(* PLC project Untitled1, Beckhoff Automation GmbH TwinCAT PLC Control 3.5.10.30 *)
(* stored: creationDateTime 2020-09-30T13:14:05.8851775, modificationDateTime 2020-09-30T13:14:05.8881769 *)

TYPE enum_E :
(
	elit_gopickup,
	elit_init0,
	elit_init1,
	elit_init2,
	elit_init3,
	elit_init4,
	elit_init5,
	elit_init6,
	elit_init7,
	elit_init8,
	elit_init9,
	elit_init_error,
	elit_init_ok,
	elit_init_sensor_check,
	elit_initialized,
	elit_running,
	elit_starting,
	elit_wait_init,
	elit_wait_start
);
END_TYPE

TYPE STATE :
STRUCT
	curTime: LREAL;
	dvar_M_example_controller_a_x2distributing AT %Q*: BOOL;
	dvar_M_example_controller_a_zdown AT %Q*: BOOL;
	dvar_M_example_controller_count AT %Q*: DINT;
	dvar_M_example_controller AT %Q*: enum_E;
	dvar_M_HardwareMap_out_a_Dstartled AT %Q*: BOOL;
	dvar_M_HardwareMap_out_a_Dresetled AT %Q*: BOOL;
	dvar_M_HardwareMap_out_a_DledQ1 AT %Q*: BOOL;
	dvar_M_HardwareMap_out_a_DledQ2 AT %Q*: BOOL;
	dvar_M_HardwareMap_out_a_Dout4 AT %Q*: BOOL;
	dvar_M_HardwareMap_out_a_Dout5 AT %Q*: BOOL;
	dvar_M_HardwareMap_out_a_Dout6 AT %Q*: BOOL;
	dvar_M_HardwareMap_out_a_Dout7 AT %Q*: BOOL;
	dvar_M_HardwareMap_out_a_pusher1 AT %Q*: BOOL;
	dvar_M_HardwareMap_out_a_pusher2 AT %Q*: BOOL;
	dvar_M_HardwareMap_out_a_pusher3 AT %Q*: BOOL;
	dvar_M_HardwareMap_out_a_Hstartled AT %Q*: BOOL;
	dvar_M_HardwareMap_out_a_Hresetled AT %Q*: BOOL;
	dvar_M_HardwareMap_out_a_HledQ1 AT %Q*: BOOL;
	dvar_M_HardwareMap_out_a_HledQ2 AT %Q*: BOOL;
	dvar_M_HardwareMap_out_a_Hout4 AT %Q*: BOOL;
	dvar_M_HardwareMap_out_a_Hout5 AT %Q*: BOOL;
	dvar_M_HardwareMap_out_a_Hout6 AT %Q*: BOOL;
	dvar_M_HardwareMap_out_a_Hout7 AT %Q*: BOOL;
	dvar_M_HardwareMap_out_a_x2distributing AT %Q*: BOOL;
	dvar_M_HardwareMap_out_a_x2testing AT %Q*: BOOL;
	dvar_M_HardwareMap_out_a_zdown AT %Q*: BOOL;
	dvar_M_HardwareMap_out_a_gripperclose AT %Q*: BOOL;
	dvar_M_HardwareMap_out_a_transfer2pickpos AT %Q*: BOOL;
	dvar_M_HardwareMap_out_a_transfer2droppos AT %Q*: BOOL;
	dvar_M_HardwareMap_out_a_vacuum AT %Q*: BOOL;
	dvar_M_HardwareMap_out_a_ejectpulse AT %Q*: BOOL;
	dvar_M_HardwareMap_out_a_handlingready AT %Q*: BOOL;
	dvar_M_HardwareMap_init_err_sen_idx AT %Q*: DINT;
	dvar_M_HardwareMap_init_err_led_idx AT %Q*: DINT;
	cvar_M_HardwareMap_t AT %Q*: LREAL;
	dvar_M_HardwareMap AT %Q*: enum_E;
END_STRUCT
END_TYPE

(* global variable list INPUTS *)
VAR_GLOBAL
	ivar_s_Dstartbutton AT %I*: BOOL;
	ivar_s_Dstopbutton AT %I*: BOOL;
	ivar_s_Dresetbutton AT %I*: BOOL;
	ivar_s_Dautoswitch AT %I*: BOOL;
	ivar_s_pusher1_in AT %I*: BOOL;
	ivar_s_pusher1_out AT %I*: BOOL;
	ivar_s_stack1filled AT %I*: BOOL;
	ivar_s_product1 AT %I*: BOOL;
	ivar_s_pusher2_in AT %I*: BOOL;
	ivar_s_pusher2_out AT %I*: BOOL;
	ivar_s_stack2filled AT %I*: BOOL;
	ivar_s_product2 AT %I*: BOOL;
	ivar_s_pusher3_in AT %I*: BOOL;
	ivar_s_pusher3_out AT %I*: BOOL;
	ivar_s_stack3filled AT %I*: BOOL;
	ivar_s_product3 AT %I*: BOOL;
	ivar_s_handlingbusy AT %I*: BOOL;
	ivar_s_Hstartbutton AT %I*: BOOL;
	ivar_s_Hstopbutton AT %I*: BOOL;
	ivar_s_Hresetbutton AT %I*: BOOL;
	ivar_s_Hautoswitch AT %I*: BOOL;
	ivar_s_xpos_at1 AT %I*: BOOL;
	ivar_s_xpos_at2 AT %I*: BOOL;
	ivar_s_xpos_at3 AT %I*: BOOL;
	ivar_s_xpos_atdrop AT %I*: BOOL;
	ivar_s_zpos_atup AT %I*: BOOL;
	ivar_s_zpos_atdown AT %I*: BOOL;
	ivar_s_gripper AT %I*: BOOL;
	ivar_s_transfer_atpickup AT %I*: BOOL;
	ivar_s_transfer_atdrop AT %I*: BOOL;
	ivar_s_transfer_athalfway AT %I*: BOOL;
	ivar_s_vacuum AT %I*: BOOL;
	ivar_s_product4 AT %I*: BOOL;
	ivar_s_testingbusy AT %I*: BOOL;
	ivar_s_Din4 AT %I*: BOOL;
	ivar_s_Din5 AT %I*: BOOL;
	ivar_s_Din6 AT %I*: BOOL;
	ivar_s_Din7 AT %I*: BOOL;
	ivar_s_Hin4 AT %I*: BOOL;
	ivar_s_Hin5 AT %I*: BOOL;
	ivar_s_Hin6 AT %I*: BOOL;
	ivar_s_Hin7 AT %I*: BOOL;
	ivar_a_Dout4 AT %I*: BOOL;
	ivar_a_Dout5 AT %I*: BOOL;
	ivar_a_Dout6 AT %I*: BOOL;
	ivar_a_Dout7 AT %I*: BOOL;
	ivar_a_Hout4 AT %I*: BOOL;
	ivar_a_Hout5 AT %I*: BOOL;
	ivar_a_Hout6 AT %I*: BOOL;
	ivar_a_Hout7 AT %I*: BOOL;
END_VAR

(* global variable list TIMERS *)
VAR_GLOBAL
	timer0: TON;
	timer1: TON;
	curTimer: INT := 0;
END_VAR

FUNCTION alg_a_DledQ1 : BOOL
VAR_INPUT
	state: STATE;
END_VAR

            alg_a_DledQ1 := FALSE;
          
END_FUNCTION

FUNCTION alg_a_DledQ2 : BOOL
VAR_INPUT
	state: STATE;
END_VAR

            alg_a_DledQ2 := FALSE;
          
END_FUNCTION

FUNCTION alg_a_Dresetled : BOOL
VAR_INPUT
	state: STATE;
END_VAR

            alg_a_Dresetled := FALSE;
          
END_FUNCTION

FUNCTION alg_a_Dstartled : BOOL
VAR_INPUT
	state: STATE;
END_VAR

            alg_a_Dstartled := alg_M_example_controller_a_Dstartled(state);
          
END_FUNCTION

FUNCTION alg_a_ejectpulse : BOOL
VAR_INPUT
	state: STATE;
END_VAR

            alg_a_ejectpulse := FALSE;
          
END_FUNCTION

FUNCTION alg_a_gripperclose : BOOL
VAR_INPUT
	state: STATE;
END_VAR

            alg_a_gripperclose := FALSE;
          
END_FUNCTION

FUNCTION alg_a_handlingready : BOOL
VAR_INPUT
	state: STATE;
END_VAR

            alg_a_handlingready := FALSE;
          
END_FUNCTION

FUNCTION alg_a_HledQ1 : BOOL
VAR_INPUT
	state: STATE;
END_VAR

            alg_a_HledQ1 := FALSE;
          
END_FUNCTION

FUNCTION alg_a_HledQ2 : BOOL
VAR_INPUT
	state: STATE;
END_VAR

            alg_a_HledQ2 := FALSE;
          
END_FUNCTION

FUNCTION alg_a_Hresetled : BOOL
VAR_INPUT
	state: STATE;
END_VAR

            alg_a_Hresetled := FALSE;
          
END_FUNCTION

FUNCTION alg_a_Hstartled : BOOL
VAR_INPUT
	state: STATE;
END_VAR

            alg_a_Hstartled := FALSE;
          
END_FUNCTION

FUNCTION alg_a_pusher1 : BOOL
VAR_INPUT
	state: STATE;
END_VAR

            alg_a_pusher1 := FALSE;
          
END_FUNCTION

FUNCTION alg_a_pusher2 : BOOL
VAR_INPUT
	state: STATE;
END_VAR

            alg_a_pusher2 := FALSE;
          
END_FUNCTION

FUNCTION alg_a_pusher3 : BOOL
VAR_INPUT
	state: STATE;
END_VAR

            alg_a_pusher3 := FALSE;
          
END_FUNCTION

FUNCTION alg_a_transfer2droppos : BOOL
VAR_INPUT
	state: STATE;
END_VAR

            alg_a_transfer2droppos := FALSE;
          
END_FUNCTION

FUNCTION alg_a_transfer2pickpos : BOOL
VAR_INPUT
	state: STATE;
END_VAR

            alg_a_transfer2pickpos := FALSE;
          
END_FUNCTION

FUNCTION alg_a_vacuum : BOOL
VAR_INPUT
	state: STATE;
END_VAR

            alg_a_vacuum := FALSE;
          
END_FUNCTION

FUNCTION alg_a_x2distributing : BOOL
VAR_INPUT
	state: STATE;
END_VAR

            alg_a_x2distributing := state.dvar_M_example_controller_a_x2distributing;
          
END_FUNCTION

FUNCTION alg_a_x2testing : BOOL
VAR_INPUT
	state: STATE;
END_VAR

            alg_a_x2testing := FALSE;
          
END_FUNCTION

FUNCTION alg_a_zdown : BOOL
VAR_INPUT
	state: STATE;
END_VAR

            alg_a_zdown := state.dvar_M_example_controller_a_zdown;
          
END_FUNCTION

FUNCTION alg_M_example_controller_a_Dstartled : BOOL
VAR_INPUT
	state: STATE;
END_VAR

            alg_M_example_controller_a_Dstartled := (state.dvar_M_example_controller) = (elit_running);
          
END_FUNCTION

FUNCTION alg_M_example_controller_godown : ARRAY[0..2] OF BOOL
VAR_INPUT
	state: STATE;
END_VAR

            alg_M_example_controller_godown := makeArray0(ivar_s_xpos_at1, ivar_s_xpos_at2, ivar_s_xpos_at3);
          
END_FUNCTION

FUNCTION alg_s_Dinitialized : BOOL
VAR_INPUT
	state: STATE;
END_VAR

            alg_s_Dinitialized := (state.dvar_M_HardwareMap) = (elit_initialized);
          
END_FUNCTION

FUNCTION alg_s_Hinitialized : BOOL
VAR_INPUT
	state: STATE;
END_VAR

            alg_s_Hinitialized := (state.dvar_M_HardwareMap) = (elit_initialized);
          
END_FUNCTION

FUNCTION derivcvar_M_HardwareMap_t : LREAL
VAR_INPUT
	state: STATE;
END_VAR

            derivcvar_M_HardwareMap_t := 1.0;
          
END_FUNCTION

PROGRAM MAIN
VAR_OUTPUT
	timerValue0: TIME;
	timerValue1: TIME;
END_VAR
VAR
	cnt: LINT;
	first: BOOL := TRUE;
	curTimerValue: TIME;
	state0: STATE;
	curTime: LREAL;
	loopsKilled: LINT;
END_VAR
VAR_TEMP
	lastTimerValue: TIME;
	curDeltaTime: TIME;
	curDeltaSecs: LREAL;
	state1: STATE;
	progress: BOOL;
	loopCount: INT;
	b1: BOOL;
	b2: BOOL;
END_VAR

            
// Handle 'time' and cycle time.
cnt := cnt + 1;

timer0(IN := curTimer = 0, PT := T#1D);
timer1(IN := curTimer = 1, PT := T#1D);
timerValue0 := timer0.ET;
timerValue1 := timer1.ET;

lastTimerValue := curTimerValue;
IF curTimer = 0 THEN
    curTimerValue := timerValue0;
ELSE
    curTimerValue := timerValue1;
END_IF;
curDeltaTime := curTimerValue - lastTimerValue;
curDeltaSecs := TIME_TO_LREAL(curDeltaTime) / 1000;
curTime := curTime + curDeltaSecs;

IF cnt MOD 10 = 0 THEN
    curTimer := 1 - curTimer;
    curTimerValue := T#0S;
    timer0(IN := curTimer = 0, PT := T#1D);
    timer1(IN := curTimer = 1, PT := T#1D);
    timerValue0 := timer0.ET;
    timerValue1 := timer1.ET;
END_IF;

IF first THEN
    first := FALSE;

    // Initialize state variables for initial state.
    state0.dvar_M_example_controller_a_x2distributing := FALSE;
    state0.dvar_M_example_controller_a_zdown := FALSE;
    state0.dvar_M_example_controller_count := 0;
    state0.dvar_M_example_controller := elit_init2;
    state0.dvar_M_HardwareMap_out_a_Dstartled := FALSE;
    state0.dvar_M_HardwareMap_out_a_Dresetled := FALSE;
    state0.dvar_M_HardwareMap_out_a_DledQ1 := TRUE;
    state0.dvar_M_HardwareMap_out_a_DledQ2 := TRUE;
    state0.dvar_M_HardwareMap_out_a_Dout4 := FALSE;
    state0.dvar_M_HardwareMap_out_a_Dout5 := FALSE;
    state0.dvar_M_HardwareMap_out_a_Dout6 := FALSE;
    state0.dvar_M_HardwareMap_out_a_Dout7 := FALSE;
    state0.dvar_M_HardwareMap_out_a_pusher1 := FALSE;
    state0.dvar_M_HardwareMap_out_a_pusher2 := FALSE;
    state0.dvar_M_HardwareMap_out_a_pusher3 := FALSE;
    state0.dvar_M_HardwareMap_out_a_Hstartled := FALSE;
    state0.dvar_M_HardwareMap_out_a_Hresetled := FALSE;
    state0.dvar_M_HardwareMap_out_a_HledQ1 := TRUE;
    state0.dvar_M_HardwareMap_out_a_HledQ2 := TRUE;
    state0.dvar_M_HardwareMap_out_a_Hout4 := FALSE;
    state0.dvar_M_HardwareMap_out_a_Hout5 := FALSE;
    state0.dvar_M_HardwareMap_out_a_Hout6 := FALSE;
    state0.dvar_M_HardwareMap_out_a_Hout7 := FALSE;
    state0.dvar_M_HardwareMap_out_a_x2distributing := TRUE;
    state0.dvar_M_HardwareMap_out_a_x2testing := TRUE;
    state0.dvar_M_HardwareMap_out_a_zdown := FALSE;
    state0.dvar_M_HardwareMap_out_a_gripperclose := FALSE;
    state0.dvar_M_HardwareMap_out_a_transfer2pickpos := FALSE;
    state0.dvar_M_HardwareMap_out_a_transfer2droppos := FALSE;
    state0.dvar_M_HardwareMap_out_a_vacuum := FALSE;
    state0.dvar_M_HardwareMap_out_a_ejectpulse := FALSE;
    state0.dvar_M_HardwareMap_out_a_handlingready := FALSE;
    state0.dvar_M_HardwareMap_init_err_sen_idx := -1;
    state0.dvar_M_HardwareMap_init_err_led_idx := 0;
    state0.cvar_M_HardwareMap_t := 0.0;
    state0.dvar_M_HardwareMap := elit_init0;
ELSE
    // Update continuous variables for time delay.
    state1.cvar_M_HardwareMap_t := state0.cvar_M_HardwareMap_t + curDeltaSecs * derivcvar_M_HardwareMap_t(state0);

    state0.curTime := curTime;
    state0.cvar_M_HardwareMap_t := state1.cvar_M_HardwareMap_t;
END_IF;

// Event loop.
WHILE TRUE DO
    progress := FALSE;

    // Event "M.example_controller_init".
    IF NOT progress THEN
        IF (state0.dvar_M_example_controller) = (elit_wait_init) THEN
            progress := TRUE;
            state1 := state0;

            state1.dvar_M_example_controller_a_x2distributing := TRUE;
            state1.dvar_M_example_controller := elit_wait_start;

            state0 := state1;
        END_IF;
    END_IF;

    // Event "M.example_controller_onpos".
    IF NOT progress THEN
        IF (state0.dvar_M_example_controller) = (elit_gopickup) THEN
            progress := TRUE;
            state1 := state0;

            state1.dvar_M_example_controller_count := (state0.dvar_M_example_controller_count) + (1);
            state1.dvar_M_example_controller_a_x2distributing := FALSE;
            state1.dvar_M_example_controller_a_zdown := TRUE;
            state1.dvar_M_example_controller := elit_running;

            state0 := state1;
        END_IF;
    END_IF;

    // Event "M.example_controller_start".
    IF NOT progress THEN
        b1 := (state0.dvar_M_example_controller) = (elit_wait_start);
        b1 := b1 AND (ivar_s_xpos_at2);
        IF b1 THEN
            progress := TRUE;
            state1 := state0;

            state1.dvar_M_example_controller_a_x2distributing := FALSE;
            state1.dvar_M_example_controller := elit_gopickup;

            state0 := state1;
        END_IF;
    END_IF;

    // Event "M.example_controller_stop".
    IF NOT progress THEN
        b1 := (state0.dvar_M_example_controller) = (elit_running);
        b1 := b1 AND (ivar_s_zpos_atup);
        IF b1 THEN
            progress := TRUE;
            state1 := state0;

            state1.dvar_M_example_controller_a_zdown := FALSE;
            state1.dvar_M_example_controller := elit_wait_start;

            state0 := state1;
        END_IF;
    END_IF;

    // Event "tau".
    IF NOT progress THEN
        b1 := (state0.dvar_M_example_controller) = (elit_init2);
        b1 := b1 AND (alg_s_Dinitialized(state0));
        IF b1 THEN
            progress := TRUE;
            state1 := state0;

            state1.dvar_M_example_controller := elit_starting;

            state0 := state1;
        END_IF;
    END_IF;

    // Event "tau".
    IF NOT progress THEN
        b1 := (state0.dvar_M_example_controller) = (elit_starting);
        b1 := b1 AND (ivar_s_Dstartbutton);
        IF b1 THEN
            progress := TRUE;
            state1 := state0;

            state1.dvar_M_example_controller := elit_wait_init;

            state0 := state1;
        END_IF;
    END_IF;

    // Event "tau".
    IF NOT progress THEN
        b1 := (state0.dvar_M_HardwareMap) = (elit_init0);
        b1 := b1 AND ((state0.cvar_M_HardwareMap_t) >= (2.0));
        IF b1 THEN
            progress := TRUE;
            state1 := state0;

            state1.dvar_M_HardwareMap := elit_init1;

            state0 := state1;
        END_IF;
    END_IF;

    // Event "tau".
    IF NOT progress THEN
        IF (state0.dvar_M_HardwareMap) = (elit_init1) THEN
            progress := TRUE;
            state1 := state0;

            state1.dvar_M_HardwareMap_out_a_x2testing := FALSE;
            state1.dvar_M_HardwareMap := elit_init2;

            state0 := state1;
        END_IF;
    END_IF;

    // Event "tau".
    IF NOT progress THEN
        b1 := (state0.dvar_M_HardwareMap) = (elit_init2);
        IF b1 THEN
            b2 := ivar_s_xpos_at1;
            b2 := b2 OR (ivar_s_xpos_at2);
            b1 := b1 AND (b2);
        END_IF;
        IF b1 THEN
            progress := TRUE;
            state1 := state0;

            state1.dvar_M_HardwareMap_out_a_x2testing := TRUE;
            state1.dvar_M_HardwareMap := elit_init3;

            state0 := state1;
        END_IF;
    END_IF;

    // Event "tau".
    IF NOT progress THEN
        IF (state0.dvar_M_HardwareMap) = (elit_init3) THEN
            progress := TRUE;
            state1 := state0;

            state1.dvar_M_HardwareMap_out_a_transfer2pickpos := TRUE;
            state1.dvar_M_HardwareMap := elit_init4;

            state0 := state1;
        END_IF;
    END_IF;

    // Event "tau".
    IF NOT progress THEN
        b1 := (state0.dvar_M_HardwareMap) = (elit_init4);
        b1 := b1 AND (ivar_s_transfer_atpickup);
        IF b1 THEN
            progress := TRUE;
            state1 := state0;

            state1.dvar_M_HardwareMap_out_a_transfer2pickpos := FALSE;
            state1.dvar_M_HardwareMap := elit_init5;

            state0 := state1;
        END_IF;
    END_IF;

    // Event "tau".
    IF NOT progress THEN
        IF (state0.dvar_M_HardwareMap) = (elit_init5) THEN
            progress := TRUE;
            state1 := state0;

            state1.dvar_M_HardwareMap_out_a_transfer2droppos := TRUE;
            state1.dvar_M_HardwareMap := elit_init6;

            state0 := state1;
        END_IF;
    END_IF;

    // Event "tau".
    IF NOT progress THEN
        b1 := (state0.dvar_M_HardwareMap) = (elit_init6);
        b1 := b1 AND (ivar_s_transfer_athalfway);
        IF b1 THEN
            progress := TRUE;
            state1 := state0;

            state1.dvar_M_HardwareMap_out_a_transfer2droppos := FALSE;
            state1.dvar_M_HardwareMap := elit_init7;

            state0 := state1;
        END_IF;
    END_IF;

    // Event "tau".
    IF NOT progress THEN
        IF (state0.dvar_M_HardwareMap) = (elit_init7) THEN
            progress := TRUE;
            state1 := state0;

            state1.dvar_M_HardwareMap_out_a_x2distributing := FALSE;
            state1.dvar_M_HardwareMap := elit_init8;

            state0 := state1;
        END_IF;
    END_IF;

    // Event "tau".
    IF NOT progress THEN
        b1 := (state0.dvar_M_HardwareMap) = (elit_init8);
        b1 := b1 AND (ivar_s_xpos_atdrop);
        IF b1 THEN
            progress := TRUE;
            state1 := state0;

            state1.dvar_M_HardwareMap_out_a_x2distributing := TRUE;
            state1.cvar_M_HardwareMap_t := 0.0;
            state1.dvar_M_HardwareMap := elit_init9;

            state0 := state1;
        END_IF;
    END_IF;

    // Event "tau".
    IF NOT progress THEN
        b1 := (state0.dvar_M_HardwareMap) = (elit_init9);
        b1 := b1 AND ((state0.cvar_M_HardwareMap_t) >= (1));
        IF b1 THEN
            progress := TRUE;
            state1 := state0;

            state1.dvar_M_HardwareMap := elit_init_sensor_check;

            state0 := state1;
        END_IF;
    END_IF;

    // Event "tau".
    IF NOT progress THEN
        b1 := (state0.dvar_M_HardwareMap) = (elit_init_sensor_check);
        b1 := b1 AND (ivar_s_Dstartbutton);
        IF b1 THEN
            progress := TRUE;
            state1 := state0;

            state1.dvar_M_HardwareMap_init_err_sen_idx := 0;
            state1.dvar_M_HardwareMap := elit_init_error;

            state0 := state1;
        END_IF;
    END_IF;

    // Event "tau".
    IF NOT progress THEN
        b1 := (state0.dvar_M_HardwareMap) = (elit_init_sensor_check);
        b1 := b1 AND (NOT(ivar_s_Dstopbutton));
        IF b1 THEN
            progress := TRUE;
            state1 := state0;

            state1.dvar_M_HardwareMap_init_err_sen_idx := 1;
            state1.dvar_M_HardwareMap := elit_init_error;

            state0 := state1;
        END_IF;
    END_IF;

    // Event "tau".
    IF NOT progress THEN
        b1 := (state0.dvar_M_HardwareMap) = (elit_init_sensor_check);
        b1 := b1 AND (ivar_s_Dautoswitch);
        IF b1 THEN
            progress := TRUE;
            state1 := state0;

            state1.dvar_M_HardwareMap_init_err_sen_idx := 2;
            state1.dvar_M_HardwareMap := elit_init_error;

            state0 := state1;
        END_IF;
    END_IF;

    // Event "tau".
    IF NOT progress THEN
        b1 := (state0.dvar_M_HardwareMap) = (elit_init_sensor_check);
        b1 := b1 AND (ivar_s_Dresetbutton);
        IF b1 THEN
            progress := TRUE;
            state1 := state0;

            state1.dvar_M_HardwareMap_init_err_sen_idx := 3;
            state1.dvar_M_HardwareMap := elit_init_error;

            state0 := state1;
        END_IF;
    END_IF;

    // Event "tau".
    IF NOT progress THEN
        b1 := (state0.dvar_M_HardwareMap) = (elit_init_sensor_check);
        b1 := b1 AND (ivar_s_Din4);
        IF b1 THEN
            progress := TRUE;
            state1 := state0;

            state1.dvar_M_HardwareMap_init_err_sen_idx := 4;
            state1.dvar_M_HardwareMap := elit_init_error;

            state0 := state1;
        END_IF;
    END_IF;

    // Event "tau".
    IF NOT progress THEN
        b1 := (state0.dvar_M_HardwareMap) = (elit_init_sensor_check);
        b1 := b1 AND (ivar_s_Din5);
        IF b1 THEN
            progress := TRUE;
            state1 := state0;

            state1.dvar_M_HardwareMap_init_err_sen_idx := 5;
            state1.dvar_M_HardwareMap := elit_init_error;

            state0 := state1;
        END_IF;
    END_IF;

    // Event "tau".
    IF NOT progress THEN
        b1 := (state0.dvar_M_HardwareMap) = (elit_init_sensor_check);
        b1 := b1 AND (ivar_s_Din6);
        IF b1 THEN
            progress := TRUE;
            state1 := state0;

            state1.dvar_M_HardwareMap_init_err_sen_idx := 6;
            state1.dvar_M_HardwareMap := elit_init_error;

            state0 := state1;
        END_IF;
    END_IF;

    // Event "tau".
    IF NOT progress THEN
        b1 := (state0.dvar_M_HardwareMap) = (elit_init_sensor_check);
        b1 := b1 AND (ivar_s_Din7);
        IF b1 THEN
            progress := TRUE;
            state1 := state0;

            state1.dvar_M_HardwareMap_init_err_sen_idx := 7;
            state1.dvar_M_HardwareMap := elit_init_error;

            state0 := state1;
        END_IF;
    END_IF;

    // Event "tau".
    IF NOT progress THEN
        b1 := (state0.dvar_M_HardwareMap) = (elit_init_sensor_check);
        b1 := b1 AND (NOT(ivar_s_pusher1_in));
        IF b1 THEN
            progress := TRUE;
            state1 := state0;

            state1.dvar_M_HardwareMap_init_err_sen_idx := 8;
            state1.dvar_M_HardwareMap := elit_init_error;

            state0 := state1;
        END_IF;
    END_IF;

    // Event "tau".
    IF NOT progress THEN
        b1 := (state0.dvar_M_HardwareMap) = (elit_init_sensor_check);
        b1 := b1 AND (ivar_s_pusher1_out);
        IF b1 THEN
            progress := TRUE;
            state1 := state0;

            state1.dvar_M_HardwareMap_init_err_sen_idx := 9;
            state1.dvar_M_HardwareMap := elit_init_error;

            state0 := state1;
        END_IF;
    END_IF;

    // Event "tau".
    IF NOT progress THEN
        b1 := (state0.dvar_M_HardwareMap) = (elit_init_sensor_check);
        b1 := b1 AND (NOT(ivar_s_stack1filled));
        IF b1 THEN
            progress := TRUE;
            state1 := state0;

            state1.dvar_M_HardwareMap_init_err_sen_idx := 10;
            state1.dvar_M_HardwareMap := elit_init_error;

            state0 := state1;
        END_IF;
    END_IF;

    // Event "tau".
    IF NOT progress THEN
        b1 := (state0.dvar_M_HardwareMap) = (elit_init_sensor_check);
        b1 := b1 AND (ivar_s_product1);
        IF b1 THEN
            progress := TRUE;
            state1 := state0;

            state1.dvar_M_HardwareMap_init_err_sen_idx := 11;
            state1.dvar_M_HardwareMap := elit_init_error;

            state0 := state1;
        END_IF;
    END_IF;

    // Event "tau".
    IF NOT progress THEN
        b1 := (state0.dvar_M_HardwareMap) = (elit_init_sensor_check);
        b1 := b1 AND (NOT(ivar_s_pusher2_in));
        IF b1 THEN
            progress := TRUE;
            state1 := state0;

            state1.dvar_M_HardwareMap_init_err_sen_idx := 12;
            state1.dvar_M_HardwareMap := elit_init_error;

            state0 := state1;
        END_IF;
    END_IF;

    // Event "tau".
    IF NOT progress THEN
        b1 := (state0.dvar_M_HardwareMap) = (elit_init_sensor_check);
        b1 := b1 AND (ivar_s_pusher2_out);
        IF b1 THEN
            progress := TRUE;
            state1 := state0;

            state1.dvar_M_HardwareMap_init_err_sen_idx := 13;
            state1.dvar_M_HardwareMap := elit_init_error;

            state0 := state1;
        END_IF;
    END_IF;

    // Event "tau".
    IF NOT progress THEN
        b1 := (state0.dvar_M_HardwareMap) = (elit_init_sensor_check);
        b1 := b1 AND (NOT(ivar_s_stack2filled));
        IF b1 THEN
            progress := TRUE;
            state1 := state0;

            state1.dvar_M_HardwareMap_init_err_sen_idx := 14;
            state1.dvar_M_HardwareMap := elit_init_error;

            state0 := state1;
        END_IF;
    END_IF;

    // Event "tau".
    IF NOT progress THEN
        b1 := (state0.dvar_M_HardwareMap) = (elit_init_sensor_check);
        b1 := b1 AND (ivar_s_product2);
        IF b1 THEN
            progress := TRUE;
            state1 := state0;

            state1.dvar_M_HardwareMap_init_err_sen_idx := 15;
            state1.dvar_M_HardwareMap := elit_init_error;

            state0 := state1;
        END_IF;
    END_IF;

    // Event "tau".
    IF NOT progress THEN
        b1 := (state0.dvar_M_HardwareMap) = (elit_init_sensor_check);
        b1 := b1 AND (NOT(ivar_s_pusher3_in));
        IF b1 THEN
            progress := TRUE;
            state1 := state0;

            state1.dvar_M_HardwareMap_init_err_sen_idx := 16;
            state1.dvar_M_HardwareMap := elit_init_error;

            state0 := state1;
        END_IF;
    END_IF;

    // Event "tau".
    IF NOT progress THEN
        b1 := (state0.dvar_M_HardwareMap) = (elit_init_sensor_check);
        b1 := b1 AND (ivar_s_pusher3_out);
        IF b1 THEN
            progress := TRUE;
            state1 := state0;

            state1.dvar_M_HardwareMap_init_err_sen_idx := 17;
            state1.dvar_M_HardwareMap := elit_init_error;

            state0 := state1;
        END_IF;
    END_IF;

    // Event "tau".
    IF NOT progress THEN
        b1 := (state0.dvar_M_HardwareMap) = (elit_init_sensor_check);
        b1 := b1 AND (NOT(ivar_s_stack3filled));
        IF b1 THEN
            progress := TRUE;
            state1 := state0;

            state1.dvar_M_HardwareMap_init_err_sen_idx := 18;
            state1.dvar_M_HardwareMap := elit_init_error;

            state0 := state1;
        END_IF;
    END_IF;

    // Event "tau".
    IF NOT progress THEN
        b1 := (state0.dvar_M_HardwareMap) = (elit_init_sensor_check);
        b1 := b1 AND (ivar_s_product3);
        IF b1 THEN
            progress := TRUE;
            state1 := state0;

            state1.dvar_M_HardwareMap_init_err_sen_idx := 19;
            state1.dvar_M_HardwareMap := elit_init_error;

            state0 := state1;
        END_IF;
    END_IF;

    // Event "tau".
    IF NOT progress THEN
        b1 := (state0.dvar_M_HardwareMap) = (elit_init_sensor_check);
        b1 := b1 AND (ivar_s_Hstartbutton);
        IF b1 THEN
            progress := TRUE;
            state1 := state0;

            state1.dvar_M_HardwareMap_init_err_sen_idx := 22;
            state1.dvar_M_HardwareMap := elit_init_error;

            state0 := state1;
        END_IF;
    END_IF;

    // Event "tau".
    IF NOT progress THEN
        b1 := (state0.dvar_M_HardwareMap) = (elit_init_sensor_check);
        b1 := b1 AND (NOT(ivar_s_Hstopbutton));
        IF b1 THEN
            progress := TRUE;
            state1 := state0;

            state1.dvar_M_HardwareMap_init_err_sen_idx := 23;
            state1.dvar_M_HardwareMap := elit_init_error;

            state0 := state1;
        END_IF;
    END_IF;

    // Event "tau".
    IF NOT progress THEN
        b1 := (state0.dvar_M_HardwareMap) = (elit_init_sensor_check);
        b1 := b1 AND (ivar_s_Hautoswitch);
        IF b1 THEN
            progress := TRUE;
            state1 := state0;

            state1.dvar_M_HardwareMap_init_err_sen_idx := 24;
            state1.dvar_M_HardwareMap := elit_init_error;

            state0 := state1;
        END_IF;
    END_IF;

    // Event "tau".
    IF NOT progress THEN
        b1 := (state0.dvar_M_HardwareMap) = (elit_init_sensor_check);
        b1 := b1 AND (ivar_s_Hresetbutton);
        IF b1 THEN
            progress := TRUE;
            state1 := state0;

            state1.dvar_M_HardwareMap_init_err_sen_idx := 25;
            state1.dvar_M_HardwareMap := elit_init_error;

            state0 := state1;
        END_IF;
    END_IF;

    // Event "tau".
    IF NOT progress THEN
        b1 := (state0.dvar_M_HardwareMap) = (elit_init_sensor_check);
        b1 := b1 AND (ivar_s_Hin4);
        IF b1 THEN
            progress := TRUE;
            state1 := state0;

            state1.dvar_M_HardwareMap_init_err_sen_idx := 26;
            state1.dvar_M_HardwareMap := elit_init_error;

            state0 := state1;
        END_IF;
    END_IF;

    // Event "tau".
    IF NOT progress THEN
        b1 := (state0.dvar_M_HardwareMap) = (elit_init_sensor_check);
        b1 := b1 AND (ivar_s_Hin5);
        IF b1 THEN
            progress := TRUE;
            state1 := state0;

            state1.dvar_M_HardwareMap_init_err_sen_idx := 27;
            state1.dvar_M_HardwareMap := elit_init_error;

            state0 := state1;
        END_IF;
    END_IF;

    // Event "tau".
    IF NOT progress THEN
        b1 := (state0.dvar_M_HardwareMap) = (elit_init_sensor_check);
        b1 := b1 AND (ivar_s_Hin6);
        IF b1 THEN
            progress := TRUE;
            state1 := state0;

            state1.dvar_M_HardwareMap_init_err_sen_idx := 28;
            state1.dvar_M_HardwareMap := elit_init_error;

            state0 := state1;
        END_IF;
    END_IF;

    // Event "tau".
    IF NOT progress THEN
        b1 := (state0.dvar_M_HardwareMap) = (elit_init_sensor_check);
        b1 := b1 AND (ivar_s_Hin7);
        IF b1 THEN
            progress := TRUE;
            state1 := state0;

            state1.dvar_M_HardwareMap_init_err_sen_idx := 29;
            state1.dvar_M_HardwareMap := elit_init_error;

            state0 := state1;
        END_IF;
    END_IF;

    // Event "tau".
    IF NOT progress THEN
        b1 := (state0.dvar_M_HardwareMap) = (elit_init_sensor_check);
        b1 := b1 AND (ivar_s_xpos_at1);
        IF b1 THEN
            progress := TRUE;
            state1 := state0;

            state1.dvar_M_HardwareMap_init_err_sen_idx := 33;
            state1.dvar_M_HardwareMap := elit_init_error;

            state0 := state1;
        END_IF;
    END_IF;

    // Event "tau".
    IF NOT progress THEN
        b1 := (state0.dvar_M_HardwareMap) = (elit_init_sensor_check);
        b1 := b1 AND (ivar_s_xpos_at2);
        IF b1 THEN
            progress := TRUE;
            state1 := state0;

            state1.dvar_M_HardwareMap_init_err_sen_idx := 34;
            state1.dvar_M_HardwareMap := elit_init_error;

            state0 := state1;
        END_IF;
    END_IF;

    // Event "tau".
    IF NOT progress THEN
        b1 := (state0.dvar_M_HardwareMap) = (elit_init_sensor_check);
        b1 := b1 AND (ivar_s_xpos_at3);
        IF b1 THEN
            progress := TRUE;
            state1 := state0;

            state1.dvar_M_HardwareMap_init_err_sen_idx := 35;
            state1.dvar_M_HardwareMap := elit_init_error;

            state0 := state1;
        END_IF;
    END_IF;

    // Event "tau".
    IF NOT progress THEN
        b1 := (state0.dvar_M_HardwareMap) = (elit_init_sensor_check);
        b1 := b1 AND (NOT(ivar_s_xpos_atdrop));
        IF b1 THEN
            progress := TRUE;
            state1 := state0;

            state1.dvar_M_HardwareMap_init_err_sen_idx := 36;
            state1.dvar_M_HardwareMap := elit_init_error;

            state0 := state1;
        END_IF;
    END_IF;

    // Event "tau".
    IF NOT progress THEN
        b1 := (state0.dvar_M_HardwareMap) = (elit_init_sensor_check);
        b1 := b1 AND (NOT(ivar_s_zpos_atup));
        IF b1 THEN
            progress := TRUE;
            state1 := state0;

            state1.dvar_M_HardwareMap_init_err_sen_idx := 37;
            state1.dvar_M_HardwareMap := elit_init_error;

            state0 := state1;
        END_IF;
    END_IF;

    // Event "tau".
    IF NOT progress THEN
        b1 := (state0.dvar_M_HardwareMap) = (elit_init_sensor_check);
        b1 := b1 AND (ivar_s_zpos_atdown);
        IF b1 THEN
            progress := TRUE;
            state1 := state0;

            state1.dvar_M_HardwareMap_init_err_sen_idx := 38;
            state1.dvar_M_HardwareMap := elit_init_error;

            state0 := state1;
        END_IF;
    END_IF;

    // Event "tau".
    IF NOT progress THEN
        b1 := (state0.dvar_M_HardwareMap) = (elit_init_sensor_check);
        b1 := b1 AND (ivar_s_gripper);
        IF b1 THEN
            progress := TRUE;
            state1 := state0;

            state1.dvar_M_HardwareMap_init_err_sen_idx := 39;
            state1.dvar_M_HardwareMap := elit_init_error;

            state0 := state1;
        END_IF;
    END_IF;

    // Event "tau".
    IF NOT progress THEN
        b1 := (state0.dvar_M_HardwareMap) = (elit_init_sensor_check);
        b1 := b1 AND (ivar_s_transfer_atpickup);
        IF b1 THEN
            progress := TRUE;
            state1 := state0;

            state1.dvar_M_HardwareMap_init_err_sen_idx := 40;
            state1.dvar_M_HardwareMap := elit_init_error;

            state0 := state1;
        END_IF;
    END_IF;

    // Event "tau".
    IF NOT progress THEN
        b1 := (state0.dvar_M_HardwareMap) = (elit_init_sensor_check);
        b1 := b1 AND (ivar_s_transfer_atdrop);
        IF b1 THEN
            progress := TRUE;
            state1 := state0;

            state1.dvar_M_HardwareMap_init_err_sen_idx := 41;
            state1.dvar_M_HardwareMap := elit_init_error;

            state0 := state1;
        END_IF;
    END_IF;

    // Event "tau".
    IF NOT progress THEN
        b1 := (state0.dvar_M_HardwareMap) = (elit_init_sensor_check);
        b1 := b1 AND (NOT(ivar_s_transfer_athalfway));
        IF b1 THEN
            progress := TRUE;
            state1 := state0;

            state1.dvar_M_HardwareMap_init_err_sen_idx := 42;
            state1.dvar_M_HardwareMap := elit_init_error;

            state0 := state1;
        END_IF;
    END_IF;

    // Event "tau".
    IF NOT progress THEN
        b1 := (state0.dvar_M_HardwareMap) = (elit_init_sensor_check);
        b1 := b1 AND (ivar_s_vacuum);
        IF b1 THEN
            progress := TRUE;
            state1 := state0;

            state1.dvar_M_HardwareMap_init_err_sen_idx := 43;
            state1.dvar_M_HardwareMap := elit_init_error;

            state0 := state1;
        END_IF;
    END_IF;

    // Event "tau".
    IF NOT progress THEN
        b1 := (state0.dvar_M_HardwareMap) = (elit_init_sensor_check);
        b1 := b1 AND (ivar_s_product4);
        IF b1 THEN
            progress := TRUE;
            state1 := state0;

            state1.dvar_M_HardwareMap_init_err_sen_idx := 44;
            state1.dvar_M_HardwareMap := elit_init_error;

            state0 := state1;
        END_IF;
    END_IF;

    // Event "tau".
    IF NOT progress THEN
        b1 := (state0.dvar_M_HardwareMap) = (elit_init_sensor_check);
        b1 := b1 AND (NOT(ivar_s_Dstartbutton));
        b1 := b1 AND (ivar_s_Dstopbutton);
        b1 := b1 AND (NOT(ivar_s_Dautoswitch));
        b1 := b1 AND (NOT(ivar_s_Dresetbutton));
        b1 := b1 AND (NOT(ivar_s_Din4));
        b1 := b1 AND (NOT(ivar_s_Din5));
        b1 := b1 AND (NOT(ivar_s_Din6));
        b1 := b1 AND (NOT(ivar_s_Din7));
        b1 := b1 AND (ivar_s_pusher1_in);
        b1 := b1 AND (NOT(ivar_s_pusher1_out));
        b1 := b1 AND (ivar_s_stack1filled);
        b1 := b1 AND (NOT(ivar_s_product1));
        b1 := b1 AND (ivar_s_pusher2_in);
        b1 := b1 AND (NOT(ivar_s_pusher2_out));
        b1 := b1 AND (ivar_s_stack2filled);
        b1 := b1 AND (NOT(ivar_s_product2));
        b1 := b1 AND (ivar_s_pusher3_in);
        b1 := b1 AND (NOT(ivar_s_pusher3_out));
        b1 := b1 AND (ivar_s_stack3filled);
        b1 := b1 AND (NOT(ivar_s_product3));
        b1 := b1 AND (NOT(ivar_s_Hstartbutton));
        b1 := b1 AND (ivar_s_Hstopbutton);
        b1 := b1 AND (NOT(ivar_s_Hautoswitch));
        b1 := b1 AND (NOT(ivar_s_Hresetbutton));
        b1 := b1 AND (NOT(ivar_s_Hin4));
        b1 := b1 AND (NOT(ivar_s_Hin5));
        b1 := b1 AND (NOT(ivar_s_Hin6));
        b1 := b1 AND (NOT(ivar_s_Hin7));
        b1 := b1 AND (NOT(ivar_s_xpos_at1));
        b1 := b1 AND (NOT(ivar_s_xpos_at2));
        b1 := b1 AND (NOT(ivar_s_xpos_at3));
        b1 := b1 AND (ivar_s_xpos_atdrop);
        b1 := b1 AND (ivar_s_zpos_atup);
        b1 := b1 AND (NOT(ivar_s_zpos_atdown));
        b1 := b1 AND (NOT(ivar_s_gripper));
        b1 := b1 AND (NOT(ivar_s_transfer_atpickup));
        b1 := b1 AND (NOT(ivar_s_transfer_atdrop));
        b1 := b1 AND (ivar_s_transfer_athalfway);
        b1 := b1 AND (NOT(ivar_s_vacuum));
        b1 := b1 AND (NOT(ivar_s_product4));
        IF b1 THEN
            progress := TRUE;
            state1 := state0;

            state1.dvar_M_HardwareMap := elit_init_ok;

            state0 := state1;
        END_IF;
    END_IF;

    // Event "tau".
    IF NOT progress THEN
        b1 := (state0.dvar_M_HardwareMap) = (elit_init_error);
        b1 := b1 AND ((state0.cvar_M_HardwareMap_t) >= (0.5));
        b1 := b1 AND ((state0.dvar_M_HardwareMap_init_err_led_idx) = (0));
        IF b1 THEN
            progress := TRUE;
            state1 := state0;

            state1.cvar_M_HardwareMap_t := 0.0;
            state1.dvar_M_HardwareMap_init_err_led_idx := 1;
            state1.dvar_M_HardwareMap_out_a_DledQ1 := TRUE;
            state1.dvar_M_HardwareMap_out_a_DledQ2 := FALSE;
            state1.dvar_M_HardwareMap_out_a_HledQ1 := TRUE;
            state1.dvar_M_HardwareMap_out_a_HledQ2 := FALSE;

            state0 := state1;
        END_IF;
    END_IF;

    // Event "tau".
    IF NOT progress THEN
        b1 := (state0.dvar_M_HardwareMap) = (elit_init_error);
        b1 := b1 AND ((state0.cvar_M_HardwareMap_t) >= (0.5));
        b1 := b1 AND ((state0.dvar_M_HardwareMap_init_err_led_idx) = (1));
        IF b1 THEN
            progress := TRUE;
            state1 := state0;

            state1.cvar_M_HardwareMap_t := 0.0;
            state1.dvar_M_HardwareMap_init_err_led_idx := 0;
            state1.dvar_M_HardwareMap_out_a_DledQ1 := FALSE;
            state1.dvar_M_HardwareMap_out_a_DledQ2 := TRUE;
            state1.dvar_M_HardwareMap_out_a_HledQ1 := FALSE;
            state1.dvar_M_HardwareMap_out_a_HledQ2 := TRUE;

            state0 := state1;
        END_IF;
    END_IF;

    // Event "tau".
    IF NOT progress THEN
        IF (state0.dvar_M_HardwareMap) = (elit_init_ok) THEN
            progress := TRUE;
            state1 := state0;

            state1.dvar_M_HardwareMap_out_a_DledQ1 := FALSE;
            state1.dvar_M_HardwareMap_out_a_DledQ2 := FALSE;
            state1.dvar_M_HardwareMap_out_a_HledQ1 := FALSE;
            state1.dvar_M_HardwareMap_out_a_HledQ2 := FALSE;
            state1.dvar_M_HardwareMap := elit_initialized;

            state0 := state1;
        END_IF;
    END_IF;

    // Event "tau".
    IF NOT progress THEN
        b1 := (state0.dvar_M_HardwareMap) = (elit_initialized);
        b1 := b1 AND ((state0.dvar_M_HardwareMap_out_a_Dstartled) <> (alg_a_Dstartled(state0)));
        IF b1 THEN
            progress := TRUE;
            state1 := state0;

            state1.dvar_M_HardwareMap_out_a_Dstartled := alg_a_Dstartled(state0);

            state0 := state1;
        END_IF;
    END_IF;

    // Event "tau".
    IF NOT progress THEN
        b1 := (state0.dvar_M_HardwareMap) = (elit_initialized);
        b1 := b1 AND ((state0.dvar_M_HardwareMap_out_a_Dresetled) <> (FALSE));
        IF b1 THEN
            progress := TRUE;
            state1 := state0;

            state1.dvar_M_HardwareMap_out_a_Dresetled := FALSE;

            state0 := state1;
        END_IF;
    END_IF;

    // Event "tau".
    IF NOT progress THEN
        b1 := (state0.dvar_M_HardwareMap) = (elit_initialized);
        b1 := b1 AND ((state0.dvar_M_HardwareMap_out_a_DledQ1) <> (FALSE));
        IF b1 THEN
            progress := TRUE;
            state1 := state0;

            state1.dvar_M_HardwareMap_out_a_DledQ1 := FALSE;

            state0 := state1;
        END_IF;
    END_IF;

    // Event "tau".
    IF NOT progress THEN
        b1 := (state0.dvar_M_HardwareMap) = (elit_initialized);
        b1 := b1 AND ((state0.dvar_M_HardwareMap_out_a_DledQ2) <> (FALSE));
        IF b1 THEN
            progress := TRUE;
            state1 := state0;

            state1.dvar_M_HardwareMap_out_a_DledQ2 := FALSE;

            state0 := state1;
        END_IF;
    END_IF;

    // Event "tau".
    IF NOT progress THEN
        b1 := (state0.dvar_M_HardwareMap) = (elit_initialized);
        b1 := b1 AND ((state0.dvar_M_HardwareMap_out_a_Dout4) <> (ivar_a_Dout4));
        IF b1 THEN
            progress := TRUE;
            state1 := state0;

            state1.dvar_M_HardwareMap_out_a_Dout4 := ivar_a_Dout4;

            state0 := state1;
        END_IF;
    END_IF;

    // Event "tau".
    IF NOT progress THEN
        b1 := (state0.dvar_M_HardwareMap) = (elit_initialized);
        b1 := b1 AND ((state0.dvar_M_HardwareMap_out_a_Dout5) <> (ivar_a_Dout5));
        IF b1 THEN
            progress := TRUE;
            state1 := state0;

            state1.dvar_M_HardwareMap_out_a_Dout5 := ivar_a_Dout5;

            state0 := state1;
        END_IF;
    END_IF;

    // Event "tau".
    IF NOT progress THEN
        b1 := (state0.dvar_M_HardwareMap) = (elit_initialized);
        b1 := b1 AND ((state0.dvar_M_HardwareMap_out_a_Dout6) <> (ivar_a_Dout6));
        IF b1 THEN
            progress := TRUE;
            state1 := state0;

            state1.dvar_M_HardwareMap_out_a_Dout6 := ivar_a_Dout6;

            state0 := state1;
        END_IF;
    END_IF;

    // Event "tau".
    IF NOT progress THEN
        b1 := (state0.dvar_M_HardwareMap) = (elit_initialized);
        b1 := b1 AND ((state0.dvar_M_HardwareMap_out_a_Dout7) <> (ivar_a_Dout7));
        IF b1 THEN
            progress := TRUE;
            state1 := state0;

            state1.dvar_M_HardwareMap_out_a_Dout7 := ivar_a_Dout7;

            state0 := state1;
        END_IF;
    END_IF;

    // Event "tau".
    IF NOT progress THEN
        b1 := (state0.dvar_M_HardwareMap) = (elit_initialized);
        b1 := b1 AND ((state0.dvar_M_HardwareMap_out_a_pusher1) <> (FALSE));
        IF b1 THEN
            progress := TRUE;
            state1 := state0;

            state1.dvar_M_HardwareMap_out_a_pusher1 := FALSE;

            state0 := state1;
        END_IF;
    END_IF;

    // Event "tau".
    IF NOT progress THEN
        b1 := (state0.dvar_M_HardwareMap) = (elit_initialized);
        b1 := b1 AND ((state0.dvar_M_HardwareMap_out_a_pusher2) <> (FALSE));
        IF b1 THEN
            progress := TRUE;
            state1 := state0;

            state1.dvar_M_HardwareMap_out_a_pusher2 := FALSE;

            state0 := state1;
        END_IF;
    END_IF;

    // Event "tau".
    IF NOT progress THEN
        b1 := (state0.dvar_M_HardwareMap) = (elit_initialized);
        b1 := b1 AND ((state0.dvar_M_HardwareMap_out_a_pusher3) <> (FALSE));
        IF b1 THEN
            progress := TRUE;
            state1 := state0;

            state1.dvar_M_HardwareMap_out_a_pusher3 := FALSE;

            state0 := state1;
        END_IF;
    END_IF;

    // Event "tau".
    IF NOT progress THEN
        b1 := (state0.dvar_M_HardwareMap) = (elit_initialized);
        b1 := b1 AND ((state0.dvar_M_HardwareMap_out_a_Hstartled) <> (FALSE));
        IF b1 THEN
            progress := TRUE;
            state1 := state0;

            state1.dvar_M_HardwareMap_out_a_Hstartled := FALSE;

            state0 := state1;
        END_IF;
    END_IF;

    // Event "tau".
    IF NOT progress THEN
        b1 := (state0.dvar_M_HardwareMap) = (elit_initialized);
        b1 := b1 AND ((state0.dvar_M_HardwareMap_out_a_Hresetled) <> (FALSE));
        IF b1 THEN
            progress := TRUE;
            state1 := state0;

            state1.dvar_M_HardwareMap_out_a_Hresetled := FALSE;

            state0 := state1;
        END_IF;
    END_IF;

    // Event "tau".
    IF NOT progress THEN
        b1 := (state0.dvar_M_HardwareMap) = (elit_initialized);
        b1 := b1 AND ((state0.dvar_M_HardwareMap_out_a_HledQ1) <> (FALSE));
        IF b1 THEN
            progress := TRUE;
            state1 := state0;

            state1.dvar_M_HardwareMap_out_a_HledQ1 := FALSE;

            state0 := state1;
        END_IF;
    END_IF;

    // Event "tau".
    IF NOT progress THEN
        b1 := (state0.dvar_M_HardwareMap) = (elit_initialized);
        b1 := b1 AND ((state0.dvar_M_HardwareMap_out_a_HledQ2) <> (FALSE));
        IF b1 THEN
            progress := TRUE;
            state1 := state0;

            state1.dvar_M_HardwareMap_out_a_HledQ2 := FALSE;

            state0 := state1;
        END_IF;
    END_IF;

    // Event "tau".
    IF NOT progress THEN
        b1 := (state0.dvar_M_HardwareMap) = (elit_initialized);
        b1 := b1 AND ((state0.dvar_M_HardwareMap_out_a_Hout4) <> (ivar_a_Hout4));
        IF b1 THEN
            progress := TRUE;
            state1 := state0;

            state1.dvar_M_HardwareMap_out_a_Hout4 := ivar_a_Hout4;

            state0 := state1;
        END_IF;
    END_IF;

    // Event "tau".
    IF NOT progress THEN
        b1 := (state0.dvar_M_HardwareMap) = (elit_initialized);
        b1 := b1 AND ((state0.dvar_M_HardwareMap_out_a_Hout5) <> (ivar_a_Hout5));
        IF b1 THEN
            progress := TRUE;
            state1 := state0;

            state1.dvar_M_HardwareMap_out_a_Hout5 := ivar_a_Hout5;

            state0 := state1;
        END_IF;
    END_IF;

    // Event "tau".
    IF NOT progress THEN
        b1 := (state0.dvar_M_HardwareMap) = (elit_initialized);
        b1 := b1 AND ((state0.dvar_M_HardwareMap_out_a_Hout6) <> (ivar_a_Hout6));
        IF b1 THEN
            progress := TRUE;
            state1 := state0;

            state1.dvar_M_HardwareMap_out_a_Hout6 := ivar_a_Hout6;

            state0 := state1;
        END_IF;
    END_IF;

    // Event "tau".
    IF NOT progress THEN
        b1 := (state0.dvar_M_HardwareMap) = (elit_initialized);
        b1 := b1 AND ((state0.dvar_M_HardwareMap_out_a_Hout7) <> (ivar_a_Hout7));
        IF b1 THEN
            progress := TRUE;
            state1 := state0;

            state1.dvar_M_HardwareMap_out_a_Hout7 := ivar_a_Hout7;

            state0 := state1;
        END_IF;
    END_IF;

    // Event "tau".
    IF NOT progress THEN
        b1 := (state0.dvar_M_HardwareMap) = (elit_initialized);
        b1 := b1 AND ((state0.dvar_M_HardwareMap_out_a_x2distributing) <> (alg_a_x2distributing(state0)));
        IF b1 THEN
            progress := TRUE;
            state1 := state0;

            state1.dvar_M_HardwareMap_out_a_x2distributing := alg_a_x2distributing(state0);

            state0 := state1;
        END_IF;
    END_IF;

    // Event "tau".
    IF NOT progress THEN
        b1 := (state0.dvar_M_HardwareMap) = (elit_initialized);
        b1 := b1 AND ((state0.dvar_M_HardwareMap_out_a_x2testing) <> (FALSE));
        IF b1 THEN
            progress := TRUE;
            state1 := state0;

            state1.dvar_M_HardwareMap_out_a_x2testing := FALSE;

            state0 := state1;
        END_IF;
    END_IF;

    // Event "tau".
    IF NOT progress THEN
        b1 := (state0.dvar_M_HardwareMap) = (elit_initialized);
        b1 := b1 AND ((state0.dvar_M_HardwareMap_out_a_zdown) <> (alg_a_zdown(state0)));
        IF b1 THEN
            progress := TRUE;
            state1 := state0;

            state1.dvar_M_HardwareMap_out_a_zdown := alg_a_zdown(state0);

            state0 := state1;
        END_IF;
    END_IF;

    // Event "tau".
    IF NOT progress THEN
        b1 := (state0.dvar_M_HardwareMap) = (elit_initialized);
        b1 := b1 AND ((state0.dvar_M_HardwareMap_out_a_gripperclose) <> (FALSE));
        IF b1 THEN
            progress := TRUE;
            state1 := state0;

            state1.dvar_M_HardwareMap_out_a_gripperclose := FALSE;

            state0 := state1;
        END_IF;
    END_IF;

    // Event "tau".
    IF NOT progress THEN
        b1 := (state0.dvar_M_HardwareMap) = (elit_initialized);
        b1 := b1 AND ((state0.dvar_M_HardwareMap_out_a_transfer2pickpos) <> (FALSE));
        IF b1 THEN
            progress := TRUE;
            state1 := state0;

            state1.dvar_M_HardwareMap_out_a_transfer2pickpos := FALSE;

            state0 := state1;
        END_IF;
    END_IF;

    // Event "tau".
    IF NOT progress THEN
        b1 := (state0.dvar_M_HardwareMap) = (elit_initialized);
        b1 := b1 AND ((state0.dvar_M_HardwareMap_out_a_transfer2droppos) <> (FALSE));
        IF b1 THEN
            progress := TRUE;
            state1 := state0;

            state1.dvar_M_HardwareMap_out_a_transfer2droppos := FALSE;

            state0 := state1;
        END_IF;
    END_IF;

    // Event "tau".
    IF NOT progress THEN
        b1 := (state0.dvar_M_HardwareMap) = (elit_initialized);
        b1 := b1 AND ((state0.dvar_M_HardwareMap_out_a_vacuum) <> (FALSE));
        IF b1 THEN
            progress := TRUE;
            state1 := state0;

            state1.dvar_M_HardwareMap_out_a_vacuum := FALSE;

            state0 := state1;
        END_IF;
    END_IF;

    // Event "tau".
    IF NOT progress THEN
        b1 := (state0.dvar_M_HardwareMap) = (elit_initialized);
        b1 := b1 AND ((state0.dvar_M_HardwareMap_out_a_ejectpulse) <> (FALSE));
        IF b1 THEN
            progress := TRUE;
            state1 := state0;

            state1.dvar_M_HardwareMap_out_a_ejectpulse := FALSE;

            state0 := state1;
        END_IF;
    END_IF;

    // Event "tau".
    IF NOT progress THEN
        b1 := (state0.dvar_M_HardwareMap) = (elit_initialized);
        b1 := b1 AND ((state0.dvar_M_HardwareMap_out_a_handlingready) <> (FALSE));
        IF b1 THEN
            progress := TRUE;
            state1 := state0;

            state1.dvar_M_HardwareMap_out_a_handlingready := FALSE;

            state0 := state1;
        END_IF;
    END_IF;

    // Done with events?
    IF NOT progress THEN
        EXIT;
    END_IF;

    // Protect against events that are always enabled.
    loopCount := loopCount + 1;
    IF loopCount >= 100 THEN
        loopsKilled := loopsKilled + 1;
        EXIT;
    END_IF;
END_WHILE;
          
END_PROGRAM

FUNCTION makeArray0 : ARRAY[0..2] OF BOOL
VAR_INPUT
	elem0: BOOL;
	elem1: BOOL;
	elem2: BOOL;
END_VAR
VAR
	rslt: ARRAY[0..2] OF BOOL;
END_VAR

            rslt[0] := elem0;
rslt[1] := elem1;
rslt[2] := elem2;
makeArray0 := rslt;
          
END_FUNCTION

FUNCTION normProjIdx : DINT
VAR_INPUT
	idx: DINT;
	size: DINT;
END_VAR
VAR
	tmp: DINT;
END_VAR

            tmp := idx;
IF tmp < 0 THEN
    tmp := size + tmp;
END_IF;
normProjIdx := tmp;
          
END_FUNCTION

FUNCTION projArray0 : BOOL
VAR_INPUT
	arr: ARRAY[0..2] OF BOOL;
	idx: DINT;
END_VAR

            projArray0 := arr[normProjIdx(idx, 3)];
          
END_FUNCTION
